(* PLC project Untitled1.project, CODESYS CODESYS V3.5 SP21 Patch 3 *)
(* stored: creationDateTime 2026-04-17T12:04:32.9281113, modificationDateTime 2025-11-16T13:06:54.2743497 *)

PROGRAM PLC_PRG
  VAR
    Level_Sim01 : Level_Sim;
    OnOff_cont_01 : OnOff_Control;
    Reset_Trig : R_TRIG;
  END_VAR

                    Reset_Trig(CLK := GVL.ResetSystem);
IF Reset_Trig.Q THEN
    // Reset all process vars to initial states
    GVL.Level_PV := 0.0;          // Tank empty
    GVL.Level_Sp := 50.0;         // Default setpoint
    GVL.Hyst := 2.0;              // Default hysteresis
    GVL.PumpCoil := FALSE;        // Pump off
    GVL.DischargeVlve := FALSE;   // Valve closed (no drain)
    GVL.AutoMode := FALSE;        // Start in manual
    GVL.SystemStart := FALSE;     // Stop system
	GVl.ResetSystem := False;
    
    // Optional: Reset internal FB states (if needed)
    // Level_Sim01.Level := 0.0;  // But Level is OUTPUT—handled via PV above
    // For deeper reset, call a custom Reset method in FBs (see Step 3)
END_IF;
IF GVL.SystemStart THEN
	GVL.DischargeVlve := TRUE;
	Level_Sim01(Charge:=GVL.PumpCoil , Discharge:=GVL.DischargeVlve , Level=>GVL.Level_PV );
	IF GVL.AutoMode THEN
		OnOff_cont_01(Feedback:=GVL.Level_PV , Setpoint:=GVL.Level_Sp , Hyst:=GVL.Hyst , ControlSig=>GVL.PumpCoil );
	END_IF
ELSE
    // Safe stop: Turn off actuators, hold level (no sim updates)
    GVL.PumpCoil := FALSE;
    GVL.DischargeVlve := FALSE;  // Assuming you want to close discharge too—adjust if it's a leak sim.
    // Optional: Reset level to 0 or SP on stop? Uncomment if needed.
    // GVL.Level_PV := 0.0;  // Or GVL.Level_Sp;
END_IF;
                  
END_PROGRAM

FUNCTION_BLOCK Level_Sim
  VAR_INPUT
    Charge : BOOL;
    Discharge : BOOL;
  END_VAR
  VAR_OUTPUT
    Level : REAL;
  END_VAR
  VAR
    Blink_Charge : Blink;
    Blink_Discharge : Blink;
    Charge_RE : R_trig;
    DisCharge_RE : R_trig;
  END_VAR

                    // Charging simulator
Blink_Charge(ENABLE:=Charge , TIMELOW:=T#100MS , TIMEHIGH:=T#100MS , OUT=> );
Charge_RE(CLK:= Blink_Charge.OUT, Q=> );
IF Charge_RE.Q THEN
	Level:= Level+0.4;
END_IF
// Discharging simulator
Blink_Discharge(ENABLE:= Discharge , TIMELOW:=T#100MS , TIMEHIGH:=T#100MS , OUT=> );
DisCharge_RE(CLK:=Blink_Discharge.OUT , Q=> );
IF DisCharge_RE.Q THEN
	Level:= Level-0.1;
END_IF
// in this case rate of charging in bigger than discharge
IF Level<0 THEN
	Level:=0;
END_IF
IF  Level > 100 THEN
	Level:=100;
END_IF



                  
END_FUNCTION_BLOCK

FUNCTION_BLOCK OnOff_Control
  VAR_INPUT
    Feedback : REAL;
    Setpoint : REAL;
    Hyst : REAL;
  END_VAR
  VAR_OUTPUT
    ControlSig : BOOL;
  END_VAR

                    IF feedback>Setpoint+Hyst/2 THEN
	ControlSig:=FALSE;
ELSIF feedback<Setpoint-Hyst/2 THEN
		ControlSig:=TRUE;
END_IF
                  
END_FUNCTION_BLOCK

CONFIGURATION Device
  RESOURCE Application ON PLC
    {attribute 'qualified_only'}
    VAR_GLOBAL  (* GVL *)
      SystemStart : BOOL := FALSE;
      AutoMode : BOOL := TRUE;
      PumpCoil : BOOL := FALSE;
      DischargeVlve : BOOL := TRUE;
      Level_PV : REAL := 0.0;
      Level_Sp : REAL := 50;
      Hyst : REAL := 2.0;
      ResetSystem : BOOL;
    END_VAR
    TASK MainTask(INTERVAL := T#20ms, PRIORITY := 1);
    PROGRAM PLC_PRG WITH MainTask : PLC_PRG;
  END_RESOURCE
END_CONFIGURATION
